(* IEC 61131-3 sources: Industry-PLC-LLM/data/PLCBEAD_repo/PLCBEAD_PLCEmbed-main/PLC-BEAD/Source/GEB/Network_IP_FIFO, 1 file *)

(* ---- IP_FIFO.ST ---- *)
TYPE
  oscat_IP_FIFO128_DATA  : ARRAY [1..128] OF BYTE;
  oscat_Mailbox  : ARRAY [1..16] OF BYTE;

  oscat_IP_FIFO_DATA :
  STRUCT
	X       : oscat_IP_FIFO128_DATA; (* IP_ID FIFO Speicher          *)
	Y       : oscat_IP_FIFO128_DATA; (* IP_ID Z�hler                 *)
	ID      : BYTE;                  (* h�chste vergabene id         *)
	MAX_ID  : BYTE;                  (* maximal Anmeldungen pro ID   *)
    INIT    : BOOL;                  (* Initialisierung durchgef�hrt *)
	EMPTY   : BOOL;                  (* FIFO leer                    *)
	FULL    : BOOL;                  (* FIFO voll                    *)
	TOP     : INT;                   (* maximale anzahl IN FIFO      *)
	NW      : INT;                   (* Schreibzeiger                *)
	NR      : INT;                   (* Lesezeiger                   *)
  END_STRUCT;
END_TYPE

TYPE

  oscat_NW_BUF_LONG  : ARRAY [0..4095] OF BYTE;

  oscat_NETWORK_BUFFER :
  STRUCT
    SIZE   : UINT;
    BUFFER : oscat_NW_BUF_LONG;
  END_STRUCT;

END_TYPE

FUNCTION _BYTE_TO_INT:INT
	VAR_INPUT
		IN :	BYTE;
	END_VAR

	_BYTE_TO_INT := USINT_TO_INT(BYTE_TO_USINT(IN));
END_FUNCTION

FUNCTION_BLOCK IP_FIFO_Block

  VAR_IN_OUT
    FIFO :	oscat_IP_FIFO_DATA;
    ID :	BYTE;
    STATE :	BYTE;
  END_VAR

  VAR
    tmp :	INT;
  END_VAR

  IF NOT FIFO.INIT THEN
    FIFO.INIT		:= TRUE;
    FIFO.NW		:= 1;
    FIFO.NR		:= 1;
    FIFO.EMPTY	:= TRUE;
    FIFO.FULL		:= FALSE;
    FIFO.TOP		:= 128;
    FIFO.MAX_ID	:= BYTE#1;
  END_IF;

  IF ID = BYTE#00 THEN
    IF FIFO.ID < INT_TO_BYTE(FIFO.TOP) THEN
      ID := USINT_TO_BYTE(BYTE_TO_USINT(FIFO.ID) + USINT#1);
      FIFO.ID := ID ;

    ELSIF STATE < BYTE#200 THEN
      STATE := BYTE#255;
    RETURN;
    END_IF;
  END_IF;

  IF STATE = BYTE#1 AND NOT FIFO.FULL THEN
    tmp := _BYTE_TO_INT(ID);
    IF FIFO.Y[tmp] < FIFO.MAX_ID THEN
      FIFO.Y[tmp] := USINT_TO_BYTE(BYTE_TO_USINT(FIFO.Y[tmp]) + USINT#1);
      tmp := FIFO.NW;
      FIFO.X[tmp] := ID;
      IF FIFO.NW = FIFO.TOP THEN FIFO.NW := 1; ELSE FIFO.NW := FIFO.NW + 1; END_IF;
      FIFO.FULL := FIFO.NW = FIFO.NR;
    FIFO.EMPTY := FALSE;
      STATE := BYTE#2;
    END_IF;
  END_IF;

  IF STATE = BYTE#2 AND NOT FIFO.EMPTY THEN
    tmp := FIFO.NR;
    IF ID = FIFO.X[tmp] THEN
      STATE := BYTE#3;
    END_IF;
  END_IF;

  IF STATE = BYTE#4 AND NOT FIFO.EMPTY THEN

    tmp := FIFO.NR;
    IF ID = FIFO.X[tmp] THEN
      tmp := _BYTE_TO_INT(ID);
      FIFO.Y[tmp] := USINT_TO_BYTE(BYTE_TO_USINT(FIFO.Y[tmp]) - USINT#1);

      IF FIFO.NR = FIFO.TOP THEN FIFO.NR := 1; ELSE FIFO.NR := FIFO.NR + 1; END_IF;
      FIFO.EMPTY := FIFO.NR = FIFO.NW;
    FIFO.FULL := FALSE;
    END_IF;
    STATE := BYTE#5;
  END_IF;

END_FUNCTION_BLOCK

PROGRAM program0
	VAR
		FIFO :	oscat_IP_FIFO_DATA;
    ID :	BYTE;
    STATE :	BYTE;

		func_block : IP_FIFO_Block;
	END_VAR
	func_block.FIFO := FIFO;
	func_block.ID := ID;
  func_block.STATE := STATE;

	func_block();
  FIFO  := func_block.FIFO;
	ID  := func_block.ID;
  STATE  := func_block.STATE;
END_PROGRAM
